PROGRAM MAIN
VAR
END_VAR

END_PROGRAM

(* stored: Version 1.1.0.1
   POU MAIN: Id {dd7b1ca3-48b8-4b4b-827b-c46336d569fa} *)
